TYPE ST_CM_SERVO :
STRUCT
	cmd: ST_CM_SERVO_CMD;
	sts: ST_CM_SERVO_STS;
END_STRUCT
END_TYPE

(* stored: Version 1.1.0.1, ProductVersion 3.1.4024.12
   DUT ST_CM_SERVO: Id {ba5de693-f086-4ea3-ae73-78a6a294ded5} *)
